FUNCTION_BLOCK FB_ServiceModule
VAR_INPUT
END_VAR
VAR_OUTPUT
	eCondition : eConditionCheck;
END_VAR
VAR
	eMode : eSystemMode;
END_VAR

PROPERTY setSLEEP : BOOL
SET
IF setSLEEP THEN
	eMode := eSystemMode.SLEEP;
ELSE
	eMode := eSystemMode.RUN;
END_IF
END_SET
END_PROPERTY

END_FUNCTION_BLOCK

(* stored: Version 1.1.0.1, ProductVersion 3.1.4024.12
   POU FB_ServiceModule: Id {c2b68249-78b4-4ae5-91f5-9de9a918b256}, SpecialFunc None
   Property setSLEEP: Id {bdce034f-f301-4cf7-92fa-495e55c34cfe}
   Set Set: Id {b4fc77e9-8c5d-4203-b030-6c6d3571f035} *)
